INTERFACE I_EventExporter

METHOD execute : BOOL
VAR_INPUT
END_VAR
END_METHOD

PROPERTY lang_code : DINT
GET
END_GET
SET
END_SET
END_PROPERTY

METHOD send_signal : BOOL
VAR_INPUT
	pAlarm		: POINTER TO FB_Alarm;
END_VAR
END_METHOD

END_INTERFACE

(* stored: Version 1.1.0.1, ProductVersion 3.1.4024.12
   Itf I_EventExporter: Id {4f3cef88-0c03-433a-a68e-c25d8f9a39f1}
   Method execute: Id {faba33dd-68ba-4f6c-9ed8-9ff726582aa0}
   Property lang_code: Id {c47c7237-b419-4941-a74d-de8f2dc1347e}
   Get Get: Id {870b92bc-bc9c-4b20-b11c-8e7308bd81a8}
   Set Set: Id {77b78c7a-9dd8-47cd-beb6-4efc406ccfd2}
   Method send_signal: Id {3d4aab7e-3102-477b-bc85-53b61297b67a} *)
